// TwinCAT 3 PLC project PLC
// ProgramVersion: 3.1.4024.0
// libraries:
//   Tc2_Standard, * (Beckhoff Automation GmbH)
//   Tc2_System, * (Beckhoff Automation GmbH)
//   Tc2_Utilities, * (Beckhoff Automation GmbH)
//   Tc3_Module, * (Beckhoff Automation GmbH)
// project tree:
//   / PlcTask.TcTTO
//   POUs/ FB_TcBSD_Backup.TcPOU, FB_TcBSD_Sendmail.TcPOU, FB_TcBSD_System.TcPOU, MAIN.TcPOU
// real-time tasks:
//   TASK PlcTask: cycle T#10ms, priority 20, ADS port 350

CONFIGURATION PLC
    RESOURCE PLC ON TwinCAT3
        TASK PlcTask(INTERVAL := T#10ms, PRIORITY := 20);
        PROGRAM MAIN WITH PlcTask : MAIN;
    END_RESOURCE
END_CONFIGURATION

// ---- POUs/MAIN.TcPOU
PROGRAM MAIN
VAR
	

//runtime counter
	iCounter:INT;
	
//system functions	
	fbTcBSD_System:FB_TcBSD_System;

//create backup
	fbTcBSD_Backup:FB_TcBSD_Backup;
	bTestBackup: BOOL;

//sendmail
	fbTcBSD_Sendmail:FB_TcBSD_Sendmail;

	
	
END_VAR

(*

-TcBSD plc tools
-permit line for Administrator -> "/usr/local/etc/doas.conf "permit nopass Administrator"


*)

//runtime control
iCounter := iCounter +1;


//backup
fbTcBSD_Backup.BackupDisk:='/dev/ada0';
fbTcBSD_Backup.BackupFolder:='/home/Administrator';
fbTcBSD_Backup.BackupName:='Backup_of_today';
fbTcBSD_Backup.Cyclic();
IF bTestBackup THEN
	bTestBackup:=FALSE;
	fbTcBSD_Backup.Execute();
END_IF

END_PROGRAM

// ---- POUs/FB_TcBSD_System.TcPOU
FUNCTION_BLOCK FB_TcBSD_System
VAR_INPUT
END_VAR
VAR_OUTPUT
END_VAR
VAR
END_VAR

END_FUNCTION_BLOCK

// ---- POUs/FB_TcBSD_Backup.TcPOU
FUNCTION_BLOCK FB_TcBSD_Backup
VAR_INPUT
END_VAR
VAR_OUTPUT
END_VAR
VAR
//SMTP Sendmail
	fbTcBackup:NT_StartProcess;			//SytemBackup
	
//Mail Sendstring
	sCommand:STRING(512);				//Command
	
//Execute
	bProcessExecute:BOOL;				//Process Execute
	bProcessActive:BOOL;				//Process Active
	bProcessBusy:BOOL;					//Process Busy
	bProcessError:BOOL;					//Process Error
	
//Bacup Parameter
	sBackupDisk:STRING;					//Backup Disk
	sBackupName:STRING;					//Backup Name
	sBackupFolder:STRING;				//backup Folder
	
//Status & Helper
	tonExecuteReset: TON;				//Timer Execute Reset
	
END_VAR

PROPERTY BackupDisk : STRING
SET
sBackupDisk:=BackupDisk;
END_SET
END_PROPERTY

PROPERTY BackupFolder : STRING
SET
sBackupFolder:=BackupFolder;
END_SET
END_PROPERTY

PROPERTY BackupName : STRING
SET
sBackupName:=BackupName;
END_SET
END_PROPERTY

METHOD BuildCommand : INT
VAR_INPUT
END_VAR
//Build Commans
sCommand:= '"TcBackup.sh --disk ';
sCommand:=CONCAT(sCommand, sBackupDisk);
sCommand:=CONCAT(sCommand, ' > ');
sCommand:=CONCAT(sCommand, sBackupFolder);
sCommand:=CONCAT(sCommand, '/');
sCommand:=CONCAT(sCommand, sBackupName);
sCommand:=CONCAT(sCommand, '.tcbkp00');
sCommand:=CONCAT(sCommand, '"');
END_METHOD

METHOD Cyclic : INT
VAR_INPUT
END_VAR
(*

--Call Cyclic

*)

BuildCommand();

//Send Mail
fbTcBackup(
	NETID:= '', 
	PATHSTR:='/bin/sh -c' , 
	DIRNAME:='/bin' , 
	COMNDLINE:=sCommand , 
	START:=bProcessActive, 
	TMOUT:= , 
	BUSY=> , 
	ERR=> , 
	ERRID=> );

//Send Execute Reset		
tonExecuteReset(IN:=bProcessExecute=FALSE AND bProcessActive=TRUE , PT:=T#5S);
IF tonExecuteReset.Q THEN
	bProcessActive:=FALSE;
END_IF
bProcessExecute:=FALSE;

//Status Signals
bProcessBusy:=bProcessActive;
IF bProcessActive AND fbTcBackup.ERR THEN
	bProcessError:=TRUE;
END_IF
END_METHOD

METHOD Execute : INT
VAR_INPUT
END_VAR
//Execute

//Build Build Command
BuildCommand();

//Flag Securtiy
if bProcessExecute=false then
	bProcessActive:=TRUE;
	bProcessError:=FALSE;
END_IF
bProcessExecute:=TRUE;
END_METHOD

END_FUNCTION_BLOCK

// ---- POUs/FB_TcBSD_Sendmail.TcPOU
FUNCTION_BLOCK FB_TcBSD_Sendmail
VAR_INPUT
END_VAR
VAR_OUTPUT
END_VAR
VAR
//SMTP Sendmail
	fbMailSend:NT_StartProcess;			//Send Mail
	
//Mail Sendstring
	sCommand:STRING(512);			//Send Command
	
//Execute Send
	bProcessExecute:BOOL;					//Send Execute
	bProcessActive:BOOL;					//Send Active
	bProcessBusy:BOOL;						//Send Busy
	bProcessError:BOOL;					//Send Error
	
//Mail Parameter
	sAddressTO:STRING;					//Mail TO
	sAddressFROM:STRING;				//Mail FROM
	sAddressCC:STRING;					//Mail CC
	sAddressBCC:STRING;					//Mail BCC
	sMailMessage:STRING(255);			//Mail Message
	sMailSubject:STRING;				//Mail Subject
	
//Status & Helper
	tonExecuteReset: TON;				//Timer Execute Reset
		
END_VAR

(*

-Send Mail with /usr/bin/mail
-Installed ssmtp package required
-v0.1

*)

PROPERTY AddressBCC : STRING
SET
sAddressBCC:=AddressBCC;
END_SET
END_PROPERTY

PROPERTY AddressCC : STRING
SET
sAddressCC:=AddressCC;
END_SET
END_PROPERTY

PROPERTY AddressFROM : STRING
SET
sAddressFROM := AddressFROM;
END_SET
END_PROPERTY

PROPERTY AddressTO : STRING
SET
sAddressTO := AddressTO;
END_SET
END_PROPERTY

METHOD PRIVATE BuildCommand : INT
VAR_INPUT
END_VAR
//Build Sendstring
sCommand:= '"echo -e ';
sCommand:=CONCAT(sCommand, '\"');
sCommand:=CONCAT(sCommand, sMailMessage);
sCommand:=CONCAT(sCommand, '\"');
sCommand:=CONCAT(sCommand, ' | ');
sCommand:=CONCAT(sCommand, 'mail -s ');
sCommand:=CONCAT(sCommand, '\"');
sCommand:=CONCAT(sCommand, sMailSubject);
sCommand:=CONCAT(sCommand, '\"');
sCommand:=CONCAT(sCommand, ' ');
sCommand:=CONCAT(sCommand, sAddressTO);
IF sAddressCC <> '' THEN
	sCommand:=CONCAT(sCommand, ' -c ');
	sCommand:=CONCAT(sCommand, sAddressCC);
END_IF
IF sAddressBCC <> '' THEN
	sCommand:=CONCAT(sCommand, ' -b ');
	sCommand:=CONCAT(sCommand, sAddressBCC);
END_IF
sCommand:=CONCAT(sCommand, ' -F');
sCommand:=CONCAT(sCommand, '\"');
sCommand:=CONCAT(sCommand, sAddressFROM);
sCommand:=CONCAT(sCommand, '\"');
sCommand:=CONCAT(sCommand, '"');
END_METHOD

METHOD Cyclic : INT
VAR_INPUT
END_VAR
(*

--Call Cyclic

*)

//Send Mail
fbMailSend(
	NETID:= '', 
	PATHSTR:='/bin/sh -c' , 
	DIRNAME:='/bin' , 
	COMNDLINE:=sCommand , 
	START:=bProcessActive, 
	TMOUT:= , 
	BUSY=> , 
	ERR=> , 
	ERRID=> );

//Send Execute Reset		
tonExecuteReset(IN:=bProcessExecute=FALSE AND bProcessActive=TRUE , PT:=T#5S);
IF tonExecuteReset.Q THEN
	bProcessActive:=FALSE;
END_IF
bProcessExecute:=FALSE;

//Status Signals
bProcessBusy:=bProcessActive;
IF bProcessActive AND fbMailSend.ERR THEN
	bProcessError:=TRUE;
END_IF
END_METHOD

METHOD PUBLIC Execute : INT
VAR_INPUT
END_VAR
//Send Mail

//Build Sendstring
BuildCommand();

//Flag Securtiy
if bProcessExecute=false then
	bProcessActive:=TRUE;
	bProcessError:=FALSE;
END_IF
bProcessExecute:=TRUE;
END_METHOD

PROPERTY MailMessage : STRING (255)
SET
sMailMessage:=MailMEssage;
END_SET
END_PROPERTY

PROPERTY MailSubject : STRING
SET
sMailSubject:=MailSubject;
END_SET
END_PROPERTY

PROPERTY SendCommand : STRING(255)
GET
SendCommand:=sCommand;
END_GET
END_PROPERTY

END_FUNCTION_BLOCK
